INTERFACE I_Machine EXTENDS I_ContainStatemachine

PROPERTY Override : LREAL
SET
END_SET
END_PROPERTY

PROPERTY Recipe : REFERENCE TO ST_Recipe
GET
END_GET
END_PROPERTY

END_INTERFACE

(* stored: Version 1.1.0.1, ProductVersion 3.1.4026.18
   Itf I_Machine: Id {fca79122-89b9-4a1f-b379-4abbced5f27b}
   Property Override: Id {c89f7003-f24c-4ee5-913c-3cbe6f23f6d5}
   Set Set: Id {4bb9dd3b-1382-4000-b75e-bf6964254785}
   Property Recipe: Id {c319658c-468c-40d5-ba0c-65e3a5df62dc}
   Get Get: Id {42edb347-818f-4d5a-975e-90e3e35a7086} *)
